FUNCTION_BLOCK Kulbana_composit
  (* Version 1.0, 2005-07-13, Goran Cengic, Chalmers *)
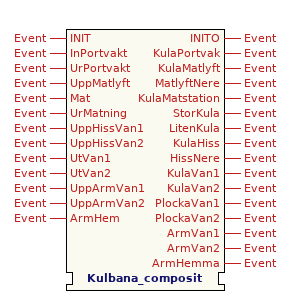
  EVENT_INPUT
    INIT;
    InPortvakt;
    UrPortvakt;
    UppMatlyft;
    Mat;
    UrMatning;
    UppHissVan1;
    UppHissVan2;
    UtVan1;
    UtVan2;
    UppArmVan1;
    UppArmVan2;
    ArmHem;
  END_EVENT
  EVENT_OUTPUT
    INITO;
    KulaPortvak;
    KulaMatlyft;
    MatlyftNere;
    KulaMatstation;
    StorKula;
    LitenKula;
    KulaHiss;
    HissNere;
    KulaVan1;
    KulaVan2;
    PlockaVan1;
    PlockaVan2;
    ArmVan1;
    ArmVan2;
    ArmHemma;
  END_EVENT
  FBS
    cycle : E_CYCLE;
    initsplit : E_SPLIT2;
    adlink : ADLINK_IO;
    split7 : E_SPLIT7;
    merge7 : E_MERGE7;
    pv : PV_model;
    ml : ML_model;
    ms : MS_model;
    msdelay : E_DELAY;
    hs : HS_model;
    vn1 : VN_model;
    vn2 : VN_model;
    ar : AR_model;
  END_FBS
  EVENT_CONNECTIONS
    INIT TO initsplit.EI;
    initsplit.EO1 TO INITO;
    initsplit.EO2 TO cycle.START;
    cycle.EO TO adlink.READ;
    adlink.VALUES TO split7.EI;
    split7.EO1 TO pv.Values;
    split7.EO2 TO ml.Values;
    split7.EO3 TO ms.Values;
    split7.EO4 TO hs.Values;
    split7.EO5 TO vn1.Values;
    split7.EO6 TO vn2.Values;
    split7.EO7 TO ar.Values;
    pv.Write TO merge7.EI1;
    ml.Write TO merge7.EI2;
    ms.Write TO merge7.EI3;
    hs.Write TO merge7.EI4;
    vn1.Write TO merge7.EI5;
    vn2.Write TO merge7.EI6;
    ar.Write TO merge7.EI7;
    merge7.EO TO adlink.WRITE;
    InPortvakt TO pv.InPortvakt;
    UrPortvakt TO pv.UrPortvakt;
    pv.KulaPortvakt TO KulaPortvakt;
    UppMatlyft TO ml.UppMatlyft;
    ml.KulaMatlyft TO KulaMatlyft;
    ml.MatlyftNere TO MatlyftNere;
    Mat TO ms.Mat;
    UrMatning TO ms.UrMatning;
    msdelay.EO TO ms.DelayDone;
    ml.KulaMatstation TO KulaMatstation;
    ml.StorKula TO StorKula;
    ml.LitenKula TO LitenKula;
    ml.Delay TO msdelay.START;
    UppHissVan1 TO hs.Mat;
    UppHissVan2 TO hs.UrMatning;
    ms.KulaHiss TO KulaHiss;
    ms.KulaVan1 TO KulaVan1;
    ms.KulaVan2 TO KulaVan2;
    ms.HissNere TO HissNere;
    UtVan1 TO vn1.UtVan;
    vn1.PlockaVan1 TO PlockaVan1;
    UtVan2 TO vn2.UtVan;
    vn2.PlockaVan2 TO PlockaVan2;
    UppArmVan1 TO ar.UppArmVan1;
    UppArmVan2 TO ar.UppArmVan2;
    ArmHem TO ar.ArmHem;
    ar.ArmVan1 TO ArmVan1;
    ar.ArmVan2 TO ArmVan2;
    ar.ArmHemma TO ArmHemma;
  END_CONNECTIONS
  DATA_CONNECTIONS
    adlink.INPUT0 TO pv.KulaPortvakt_sig;
    pv.InPortvakt_sig TO adlink.OUTPUT0;
    pv.UrPortvakt_sig TO adlink.OUTPUT1;
    adlink.INPUT TO ml.MatlyftNere_sig;
    adlink.INPUT TO ml.KulaMatlyft_sig;
    adlink.INPUT TO ml.MatlyftUppe_sig;
    adlink.INPUT TO ml.KulaMatstation_sig;
    ml.UppMatlyft_sig TO adlink.OUTPUT;
    adlink.INPUT TO ms.KulaMatstation_sig;
    adlink.INPUT TO ms.StorKula_sig;
    adlink.INPUT TO ms.LitenKula_sig;
    ms.Mat_sig TO adlink.OUTPUT;
    ms.UrMatning_sig TO adlink.OUTPUT;
    200 TO msdelay.DT;
    adlink.INPUT TO hs.HissNere_sig;
    adlink.INPUT TO hs.KulaHiss_sig;
    adlink.INPUT TO hs.HissVan1_sig;
    adlink.INPUT TO hs.KulaVan1_sig;
    adlink.INPUT TO hs.HissVan2_sig;
    adlink.INPUT TO hs.KulaVan2_sig;
    hs.UppHissVan1_sig TO adlink.OUTPUT;
    hs.UppHissVan2_sig TO adlink.OUTPUT;
    adlink.INPUT TO vn1.KulaVan_sig;
    adlink.INPUT TO vn1.PlockaVan_sig;
    adlink.INPUT TO vn1.KulaFast_sig;
    adlink.INPUT TO vn1.ArmVan_sig;
    adlink.INPUT TO vn1.ArmHemma_sig;
    vn1.UtVan_sig TO adlink.OUTPUT;
    vn1.LyftVan_sig TO adlink.OUTPUT;
    adlink.INPUT TO vn2.KulaVan_sig;
    adlink.INPUT TO vn2.PlockaVan_sig;
    adlink.INPUT TO vn2.KulaFast_sig;
    adlink.INPUT TO vn2.ArmVan_sig;
    adlink.INPUT TO vn2.ArmHemma_sig;
    vn2.UtVan_sig TO adlink.OUTPUT;
    vn2.LyftVan_sig TO adlink.OUTPUT;
    adlink.INPUT TO ar.ArmVan1_sig;
    adlink.INPUT TO ar.ArmVan2_sig;
    adlink.INPUT TO ar.KulaFast_sig;
    adlink.INPUT TO ar.ArmHemma_sig;
    ar.UppArmVan1_sig TO adlink.OUTPUT;
    ar.UppArmVan2_sig TO adlink.OUTPUT;
    ar.VridArmHoger_sig TO adlink.OUTPUT;
    ar.Sug_sig TO adlink.OUTPUT;
  END_CONNECTIONS
END_FUNCTION_BLOCK
(* other elements stored in the file *)
(* Values split *)
(* Write merge *)
(* Portvakt *)
(* Matlyft *)
(* Matstation *)
(* Hiss *)
(* Vaning 1 *)
(* Vaning 2 *)
(* Arm *)
(* Connection Source="500" Destination="cycle.DT" / *)
(* Portvakt signals *)
(* Matlyft signals *)
(* Matstation signals *)
(* Hiss signal *)
(* Vaning 1 signals *)
(* Vaning 2 signals *)
(* Arm signals *)
